// TIA Portal V20 export
FUNCTION "OPmode_01" : Void   // FC2, LAD
{ S7_Optimized_Access := 'TRUE' }
// stored: SetENOAutomatically false
BEGIN

REGION Network 1
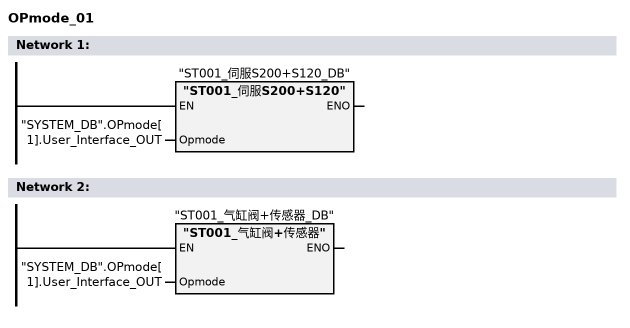
   RUNG wire#powerrail
      "ST001_伺服S200+S120_DB"(Opmode := "SYSTEM_DB".OPmode[1].User_Interface_OUT)
   END_RUNG
   // the same network as SCL:
   "ST001_伺服S200+S120_DB"(Opmode := "SYSTEM_DB".OPmode[1].User_Interface_OUT);   // "ST001_伺服S200+S120"
END_REGION

REGION Network 2
   RUNG wire#powerrail
      "ST001_气缸阀+传感器_DB"(Opmode := "SYSTEM_DB".OPmode[1].User_Interface_OUT)
   END_RUNG
   // the same network as SCL:
   "ST001_气缸阀+传感器_DB"(Opmode := "SYSTEM_DB".OPmode[1].User_Interface_OUT);   // "ST001_气缸阀+传感器"
END_REGION
END_FUNCTION
